(*********************************** G.D S.p.A. - Technical Department ***********************************
============= PROGRAM INFO ============
FOLDER:             TBD
MACHINES INVOLVED:  TBD 

============= DESCRIPTION =============
csp brand management program

============= REVISIONS ===============
Date		Version	 	Author      	Description             
----------	-------		------------  	--------------------------------------------
2019/04/05 	0000.00	 	M.Grasso		Creation of the PRG

**********************************************************************************************************)
(*$R
	process_ref := prc;
$*)
PROGRAM csp_transfer_main_brand
VAR
	prc:														process;
	prc_path:													STRING;

	cam_data_changed:											BOOL;	
		
END_VAR

_read_var_input();

_object_manager();

IF NOT objects_running()
THEN
	RETURN;	
END_IF

_read_process_image();

_mode_manager();

CASE process_get_mode(prc) OF
	MODE_ABSENT,
	MODE_INACTIVE:
		RETURN;
	MODE_TEST:
		_handle_process_test();
END_CASE

_set_runtime_properties();

(********************************* BODY *********************************)

cam_data_changed := csp_main_accuchange.cam_data_changed;

(************************************************************************)

_handle_messages();

_write_output();

ACTION _handle_messages:
;
END_ACTION

ACTION _handle_process_test:
;
END_ACTION

ACTION _mode_manager:
IF process_mode_req_is_pending(prc)
THEN
    process_apply_mode_req_first_step(prc);
    CASE process_get_mode(prc) OF
        MODE_TO_ABSENT:
			;
        MODE_TO_INACTIVE:
			;
        MODE_TO_TEST:
			;
        MODE_TO_OPERATIONAL:
			;
    END_CASE
    process_apply_mode_req_second_step(prc);
END_IF
END_ACTION

ACTION _object_manager:
IF objects_initialization()
THEN
	sub_process_init(
		object_name					:= 'csp_transfer_main_brand.prc', 
		process						:= csp_transfer_main.prc, 
		CONVERSION_this				:= prc);
		
	prc_path 						:= process_get_path(prc);
END_IF

IF objects_running()
THEN
	process_cycle(prc);
END_IF
END_ACTION

ACTION _read_process_image:
;
END_ACTION

ACTION _read_var_input:
;
END_ACTION

ACTION _set_runtime_properties:
;
END_ACTION

ACTION _write_output:
;
END_ACTION

END_PROGRAM

(* stored: Version 1.1.0.1, ProductVersion 3.1.4024.3
   POU csp_transfer_main_brand: Id {82674882-91dd-4ec6-9fe7-e558923203ef}, SpecialFunc None
   Action _handle_messages: Id {3442cc70-526d-4a9a-95f4-59728c58db5b}
   Action _handle_process_test: Id {473e0327-e52b-4208-b1db-52db50dbbc0c}
   Action _mode_manager: Id {3fc03608-a046-4cd4-9e24-8253217dadbd}
   Action _object_manager: Id {d062042c-169a-4847-b167-ace6508e0166}
   Action _read_process_image: Id {b0901103-da5a-48c3-aae3-e23185caa511}
   Action _read_var_input: Id {239193d1-1548-4f4c-9ca2-8f270bd30b34}
   Action _set_runtime_properties: Id {77acbb5b-c43a-454c-859b-0c3e6faf77bb}
   Action _write_output: Id {07ad9aae-0b0f-4380-b641-b6dc0f563511} *)
